TYPE SafetyIOParts :
STRUCT
	///DA: Dome access I/O
	domeAccess: SafetyDomeAccessIO;
	///HS: Hydraulics and Safety I/O
	hydraulicsAndSafety: SafetyHydraulicsAndSafetyIO;
END_STRUCT
END_TYPE

(* stored: Version 1.1.0.1, ProductVersion 3.1.4019.2
   DUT SafetyIOParts: Id {78de5453-057d-457f-8942-5229483af652} *)
